// TwinCAT 3 PLC project crane_program_HMI
// ProgramVersion: 3.1.4023.0
// libraries:
//   Tc2_Standard, * (Beckhoff Automation GmbH)
//   Tc2_System, * (Beckhoff Automation GmbH)
//   Tc3_Module, * (Beckhoff Automation GmbH)
// project tree:
//   / GlobalTextList.TcGTLO, PlcTask.TcTTO, Visualization Manager.TcVMO (not stored)
//   GVLs/ input.TcGVL, output.TcGVL, parameter.TcGVL
//   POUs/ MAIN.TcPOU
//   VISUs/ CraneHMI.TcVIS
// real-time tasks:
//   TASK PlcTask: cycle T#10ms, priority 20, ADS port 350

CONFIGURATION crane_program_HMI
    RESOURCE PLC ON TwinCAT3
        TASK PlcTask(INTERVAL := T#10ms, PRIORITY := 20);
        PROGRAM MAIN WITH PlcTask : MAIN;
    END_RESOURCE
END_CONFIGURATION

// ---- GVLs/input.TcGVL
{attribute 'qualified_only'}
VAR_GLOBAL
	bEnableSwitch : BOOL;
	bModeSwitch : BOOL;
	bStartSwitch : BOOL;
	
	


END_VAR

// ---- GVLs/output.TcGVL
{attribute 'qualified_only'}
VAR_GLOBAL
	bRunningLight : BOOL;
	fCylinderStroke : REAL;
	fCylinderVelocity : REAL;
	fTimeInSeconds : REAL;
END_VAR

// ---- GVLs/parameter.TcGVL
{attribute 'qualified_only'}
VAR_GLOBAL
	fCycleTime : REAL := 0.01;
	fRefCylinderVelocity : REAL;
	fRefCylinderStroke : REAL;
	iMaxCylinderStroke : INT := 2;
	iMinCylinderStroke : INT := 0;
	fAutoTime : REAL;
END_VAR

// ---- POUs/MAIN.TcPOU
PROGRAM MAIN
VAR
END_VAR

IF input.bEnableSwitch = FALSE THEN
	input.bStartSwitch := FALSE;
END_IF

IF input.bStartSwitch = TRUE THEN
	output.bRunningLight := TRUE;
	output.fTimeInSeconds := output.fTimeInSeconds + parameter.fCycleTime;
ELSE
	output.bRunningLight := FALSE;
	output.fTimeInSeconds := 0;
END_IF

IF output.bRunningLight = TRUE AND input.bModeSwitch = TRUE THEN
	output.fCylinderStroke := parameter.fRefCylinderStroke;
ELSIF output.bRunningLight = TRUE AND input.bModeSwitch = FALSE 
AND parameter.iMinCylinderStroke <= output.fCylinderStroke 
AND output.fCylinderStroke <= parameter.iMaxCylinderStroke THEN
	output.fCylinderVelocity := parameter.fRefCylinderVelocity;
	parameter.fAutoTime := parameter.fAutoTime + parameter.fCycleTime;
	output.fCylinderStroke := output.fCylinderVelocity * parameter.fAutoTime;
	IF output.fCylinderStroke <= parameter.iMinCylinderStroke 
	OR output.fCylinderStroke >= parameter.iMaxCylinderStroke THEN
		parameter.fAutoTime := 0;
	END_IF
END_IF

END_PROGRAM

// ---- GlobalTextList.TcGTLO
TEXTLIST GlobalTextList
  333 = 'AUTO'
  96 = 'ENABLE'
  840 = 'Manual'
  163 = 'MANUAL'
  746 = 'MODE'
  431 = 'RUNNING'
  835 = 'START'
END_TEXTLIST

// ---- VISUs/CraneHMI.TcVIS
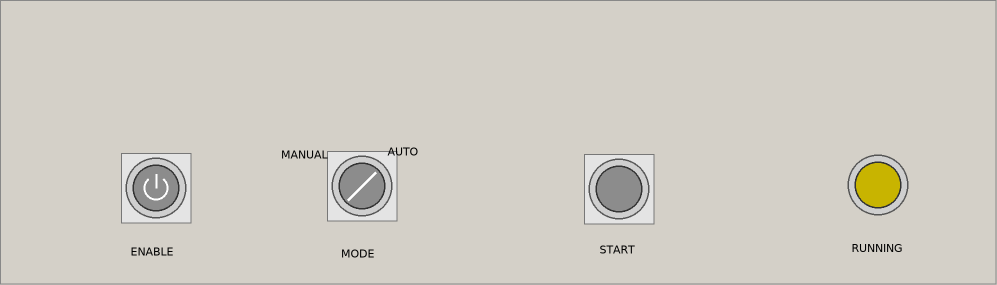
VISUALIZATION CraneHMI  // 997x285
    Lamp1 (843,150 70x70), style: Lamp-Lamp1-Yellow
    PowerSwitch (121,153 70x70), behaviour: TOGGLE, style: Switch-PowerSwitch-Gray
    RotarySwitch (327,151 70x70), behaviour: TOGGLE, style: Switch-RotarySwitch-Gray
    PushSwitch (584,154 70x70), behaviour: TOGGLE, style: Switch-PushSwitch-Gray
    Label (757,220 240x57), "RUNNING"
    Label (224,223 268x62), "MODE"
    Label (77,237 150x30), "ENABLE"
    Label (542,235 150x30), "START"
    Label (252,136 105x38), "MANUAL"
    Label (315,120 176x64), "AUTO"
END_VISUALIZATION
